PROGRAM PRG_TEST
VAR
    fbSum_Test : FB_Sum_Test; // This is our test suite
END_VAR

TcUnit.RUN();

END_PROGRAM

(* stored: Version 1.1.0.1, ProductVersion 3.1.4024.12
   POU PRG_TEST: Id {af7480f4-ba3c-4661-9624-3fca8a7e8550}, SpecialFunc None *)
